// TIA Portal V21 export
DATA_BLOCK "Ksd1"   // DB6
// stored: InstanceOfName ConeCrusher, InstanceOfType FB
"ConeCrusher"
   // VAR_INPUT
   //    sysTime : Time;
   //    resetBlock : Bool;
   //    parentRefDesignator : WString;
   //    crusherBtnStartRaw : Bool;
   //    crusherBtnStopRaw : Bool;
   //    crusherKeySwitchRaw : Bool;
   //    crusherEmStopRaw : Bool;
   //    crusherBtnResetRaw : Bool;
   //    crusherBtnStartLuSRaw : Bool;
   //    crusherBtnStopLuSRaw : Bool;
   //    premoldingSwRaw : Bool;
   //    prestartAlmFbRaw : Bool;
   //    sgReadyRaw : Bool;
   //    sgFbOnRaw : Bool;
   //    sgFbOffRaw : Bool;
   //    crusherEccentricTempRaw : Int;
   //    crusherOuterBearingTempRaw : Int;
   //    crusherInnerBearingTempRaw : Int;
   //    driveFrontBearingTempRaw : Int;
   //    driveRearBearingTempRaw : Int;
   //    driveWindingTempP1Raw : Int;
   //    driveWindingTempP2Raw : Int;
   //    driveWindingTempP3Raw : Int;
   //    driveCurrentRaw : Int;
   //    luSLocalModeSwitchRaw : Bool;
   //    luSBtnStartRaw : Bool;
   //    luSBtnStopRaw : Bool;
   //    luSBtnResetRaw : Bool;
   //    oilPump1SelSwitchRaw : Bool;
   //    oilPump2SelSwitchRaw : Bool;
   //    oilPreparationSwitchRaw : Bool;
   //    returnOilFlowSwitchRaw : Bool;
   //    oilLevelMaxRaw : Bool;
   //    oilLevelMidRaw : Bool;
   //    oilLevelMinRaw : Bool;
   //    oilTempSwitchHighRaw : Bool;
   //    oilTempSwitchLowRaw : Bool;
   //    fbPump1Raw : Bool;
   //    fbPump2Raw : Bool;
   //    pump1FaultRaw : Bool;
   //    pump2FaultRaw : Bool;
   //    oilTempTankRaw : Int;
   //    returnOilTempRaw : Int;
   //    oilFlowRaw : Int;
   //    inletWaterTemperatureRaw : Int;
   //    outletWaterTemperatureRaw : Int;
   //    inletOilTemperatureRaw : Int;
   //    inletOilPressureRaw : Int;
   // END_VAR
   // VAR_OUTPUT
   //    sgStartRaw : Bool;
   //    sgStopRaw : Bool;
   //    preStartAlmOnRaw : Bool;
   //    feedEnRaw : Bool;
   //    pump1StartRaw : Bool;
   //    pump2StartRaw : Bool;
   //    heaterOnRaw : Bool;
   //    waterVlvOpenRaw : Bool;
   //    oilToCoolerVlvRaw : Bool;
   // END_VAR
   // VAR_IN_OUT
   //    IO : "coneCrusherIOs";
   //    cfg : "coneCrusherConfigs";
   //    hmi : "coneCrusherHMIs";
   //    simHmi : "coneCrusherSimHMI";
   // END_VAR
   // VAR
   //    modelTimer : Time;
   //    prevSysTime : Time;
   //    crusher { S7_SetPoint := 'True'} : "ConeCrusherControl";
   //    crusherModel { S7_SetPoint := 'True'} : "ConeCrusherSim";
   //    crusherBtnStart { S7_SetPoint := 'True'} : "LBC_DigitalSignal";
   //    crusherBtnStop { S7_SetPoint := 'True'} : "LBC_DigitalSignal";
   //    crusherKeySwitch { S7_SetPoint := 'True'} : "LBC_DigitalSignal";
   //    crusherEmStop { S7_SetPoint := 'True'} : "LBC_DigitalSignal";
   //    crusherBtnReset { S7_SetPoint := 'True'} : "LBC_DigitalSignal";
   //    crusherBtnStartLuS { S7_SetPoint := 'True'} : "LBC_DigitalSignal";
   //    crusherBtnStopLuS { S7_SetPoint := 'True'} : "LBC_DigitalSignal";
   //    premoldingSw { S7_SetPoint := 'True'} : "LBC_DigitalSignal";
   //    prestartAlmFb { S7_SetPoint := 'True'} : "LBC_DigitalSignal";
   //    sgReady { S7_SetPoint := 'True'} : "LBC_DigitalSignal";
   //    sgFbOn { S7_SetPoint := 'True'} : "LBC_DigitalSignal";
   //    sgFbOff { S7_SetPoint := 'True'} : "LBC_DigitalSignal";
   //    crusherEccentricTemp { S7_SetPoint := 'True'} : "LBC_AnalogInput";
   //    crusherOuterBearingTemp { S7_SetPoint := 'True'} : "LBC_AnalogInput";
   //    crusherInnerBearingTemp { S7_SetPoint := 'True'} : "LBC_AnalogInput";
   //    driveFrontBearingTemp { S7_SetPoint := 'True'} : "LBC_AnalogInput";
   //    driveRearBearingTemp { S7_SetPoint := 'True'} : "LBC_AnalogInput";
   //    driveWindingTempP1 { S7_SetPoint := 'True'} : "LBC_AnalogInput";
   //    driveWindingTempP2 { S7_SetPoint := 'True'} : "LBC_AnalogInput";
   //    driveWindingTempP3 { S7_SetPoint := 'True'} : "LBC_AnalogInput";
   //    driveCurrent { S7_SetPoint := 'True'} : "LBC_AnalogInput";
   //    sgStart { S7_SetPoint := 'True'} : "LBC_DigitalSignal";
   //    sgStop { S7_SetPoint := 'True'} : "LBC_DigitalSignal";
   //    preStartAlmOn { S7_SetPoint := 'True'} : "LBC_DigitalSignal";
   //    feedEn { S7_SetPoint := 'True'} : "LBC_DigitalSignal";
   //    luSLocalModeSwitch { S7_SetPoint := 'True'} : "LBC_DigitalSignal";
   //    luSBtnStart { S7_SetPoint := 'True'} : "LBC_DigitalSignal";
   //    luSBtnStop { S7_SetPoint := 'True'} : "LBC_DigitalSignal";
   //    luSBtnReset { S7_SetPoint := 'True'} : "LBC_DigitalSignal";
   //    oilPump1SelSwitch { S7_SetPoint := 'True'} : "LBC_DigitalSignal";
   //    oilPump2SelSwitch { S7_SetPoint := 'True'} : "LBC_DigitalSignal";
   //    oilPreparationSwitch { S7_SetPoint := 'True'} : "LBC_DigitalSignal";
   //    returnOilFlowSwitch { S7_SetPoint := 'True'} : "LBC_DigitalSignal";
   //    oilLevelMax { S7_SetPoint := 'True'} : "LBC_DigitalSignal";
   //    oilLevelMid { S7_SetPoint := 'True'} : "LBC_DigitalSignal";
   //    oilLevelMin { S7_SetPoint := 'True'} : "LBC_DigitalSignal";
   //    oilTempSwitchHigh { S7_SetPoint := 'True'} : "LBC_DigitalSignal";
   //    oilTempSwitchLow { S7_SetPoint := 'True'} : "LBC_DigitalSignal";
   //    fbPump1 { S7_SetPoint := 'True'} : "LBC_DigitalSignal";
   //    fbPump2 { S7_SetPoint := 'True'} : "LBC_DigitalSignal";
   //    pump1Fault { S7_SetPoint := 'True'} : "LBC_DigitalSignal";
   //    pump2Fault { S7_SetPoint := 'True'} : "LBC_DigitalSignal";
   //    oilTempTank { S7_SetPoint := 'True'} : "LBC_AnalogInput";
   //    returnOilTemp { S7_SetPoint := 'True'} : "LBC_AnalogInput";
   //    oilFlow { S7_SetPoint := 'True'} : "LBC_AnalogInput";
   //    inletWaterTemperature { S7_SetPoint := 'True'} : "LBC_AnalogInput";
   //    outletWaterTemperature { S7_SetPoint := 'True'} : "LBC_AnalogInput";
   //    inletOilTemperature { S7_SetPoint := 'True'} : "LBC_AnalogInput";
   //    inletOilPressure { S7_SetPoint := 'True'} : "LBC_AnalogInput";
   //    pump1Start { S7_SetPoint := 'True'} : "LBC_DigitalSignal";
   //    pump2Start { S7_SetPoint := 'True'} : "LBC_DigitalSignal";
   //    heaterOn { S7_SetPoint := 'True'} : "LBC_DigitalSignal";
   //    waterVlvOpen { S7_SetPoint := 'True'} : "LBC_DigitalSignal";
   //    oilToCoolerVlv { S7_SetPoint := 'True'} : "LBC_DigitalSignal";
   // END_VAR
BEGIN
END_DATA_BLOCK
